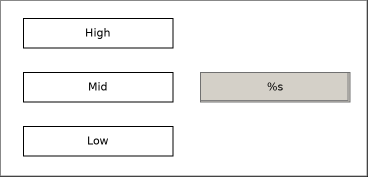
VISUALIZATION FloorVisu  // 368x177
VAR_IN_OUT
	Callbt	:	BOOL;
	Low,Mid,High	:	BOOL;
	name:STRING;
END_VAR
    Rectangle (0,0 368x177)
    Button (200,72 150x30), "%s", text variable: name
        tap Callbt
    Rectangle (23,126 150x30), "Low"
        tap Low
    Rectangle (23,72 150x30), "Mid"
        tap Mid
    Rectangle (23,18 150x30), "High"
        tap High
END_VISUALIZATION

(* stored: Version 1.1.0.1, ProductVersion 3.1.4024.9
   Visu FloorVisu: Id {f1bde99f-b1a1-4cb3-93ba-6c08fcf1b410} *)
